FUNCTION_BLOCK ACMotor
VAR
	moveContactor : ContactorNO;
END_VAR

PROPERTY IsMoving : BOOL
GET
IsMoving := moveContactor.IsClosed;
END_GET
END_PROPERTY

METHOD Start
VAR_INPUT
END_VAR
moveContactor.Close();
END_METHOD

METHOD Stop
VAR_INPUT
END_VAR
moveContactor.Open();
END_METHOD

END_FUNCTION_BLOCK

(* stored: Version 1.1.0.1, ProductVersion 3.1.4024.12
   POU ACMotor: Id {18b835c4-e8ec-487b-8a92-cd68cf60248b}, SpecialFunc None
   Property IsMoving: Id {91f61c3e-0fcd-44f7-b290-388e366d0c01}
   Get Get: Id {e49b438c-fba6-458c-b140-94eaf0057913}
   Method Start: Id {cc77df1d-29c6-466e-99ad-a6f75d0501e3}
   Method Stop: Id {5374ec64-6cb3-4288-b860-f298d3e560fb} *)
